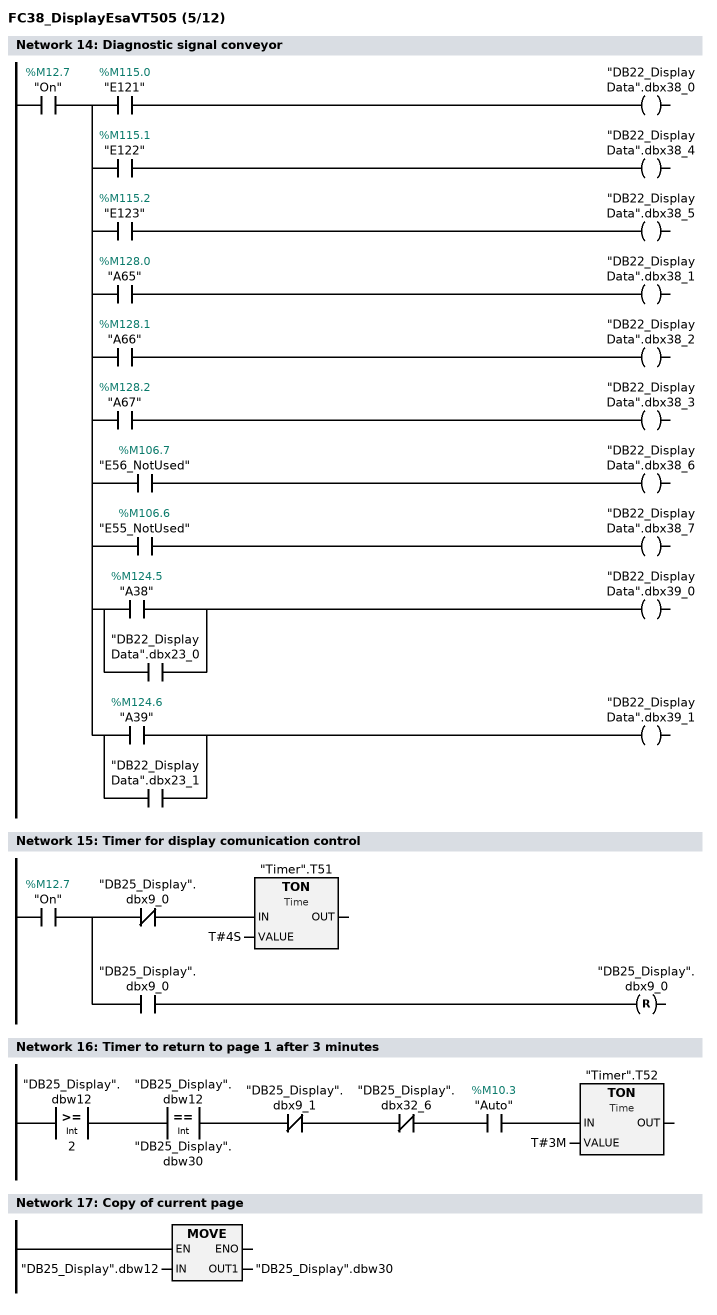
   RUNG wire#powerrail
      Contact( "On" )
      wire#w1
      Contact( "E121" )
      Coil( "DB22_DisplayData".dbx38_0 )
   END_RUNG
   RUNG wire#w1
      Contact( "E122" )
      Coil( "DB22_DisplayData".dbx38_4 )
   END_RUNG
   RUNG wire#w1
      Contact( "E123" )
      Coil( "DB22_DisplayData".dbx38_5 )
   END_RUNG
   RUNG wire#w1
      Contact( "A65" )
      Coil( "DB22_DisplayData".dbx38_1 )
   END_RUNG
   RUNG wire#w1
      Contact( "A66" )
      Coil( "DB22_DisplayData".dbx38_2 )
   END_RUNG
   RUNG wire#w1
      Contact( "A67" )
      Coil( "DB22_DisplayData".dbx38_3 )
   END_RUNG
   RUNG wire#w1
      Contact( "E56_NotUsed" )
      Coil( "DB22_DisplayData".dbx38_6 )
   END_RUNG
   RUNG wire#w1
      Contact( "E55_NotUsed" )
      Coil( "DB22_DisplayData".dbx38_7 )
   END_RUNG
   RUNG wire#w1
      Contact( "A38" )
      wire#w2
      Coil( "DB22_DisplayData".dbx39_0 )
   END_RUNG
   RUNG wire#w1
      Contact( "DB22_DisplayData".dbx23_0 )
   END_RUNG wire#w2
   RUNG wire#w1
      Contact( "A39" )
      wire#w3
      Coil( "DB22_DisplayData".dbx39_1 )
   END_RUNG
   RUNG wire#w1
      Contact( "DB22_DisplayData".dbx23_1 )
   END_RUNG wire#w3
   // the same network as SCL:
   "DB22_DisplayData".dbx38_0 := "On" AND "E121";
   "DB22_DisplayData".dbx38_4 := "On" AND "E122";
   "DB22_DisplayData".dbx38_5 := "On" AND "E123";
   "DB22_DisplayData".dbx38_1 := "On" AND "A65";
   "DB22_DisplayData".dbx38_2 := "On" AND "A66";
   "DB22_DisplayData".dbx38_3 := "On" AND "A67";
   "DB22_DisplayData".dbx38_6 := "On" AND "E56_NotUsed";
   "DB22_DisplayData".dbx38_7 := "On" AND "E55_NotUsed";
   "DB22_DisplayData".dbx39_0 := "On" AND ("A38" OR "DB22_DisplayData".dbx23_0);
   "DB22_DisplayData".dbx39_1 := "On" AND ("A39" OR "DB22_DisplayData".dbx23_1);
END_REGION

REGION Network 15: Timer for display comunication control
   "Timer".T51.TON(IN := "On" AND NOT "DB25_Display".dbx9_0, PT := T#4S);   // TON coil
   IF "On" AND "DB25_Display".dbx9_0 THEN "DB25_Display".dbx9_0 := FALSE; END_IF;
END_REGION

REGION Network 16: Timer to return to page 1 after 3 minutes
   "Timer".T52.TON(IN := ("DB25_Display".dbw12 >= 2) AND ("DB25_Display".dbw12 = "DB25_Display".dbw30) AND NOT "DB25_Display".dbx9_1 AND NOT "DB25_Display".dbx32_6 AND "Auto", PT := T#3M);   // TON coil
END_REGION

REGION Network 17: Copy of current page
   RUNG wire#powerrail
      { S7_GenerateENO := "TRUE" } Move(in := "DB25_Display".dbw12, out1 => "DB25_Display".dbw30)
   END_RUNG
   // the same network as SCL:
   "DB25_Display".dbw30 := "DB25_Display".dbw12;
END_REGION

REGION Network 18: Return to page 1 after 3 minutes
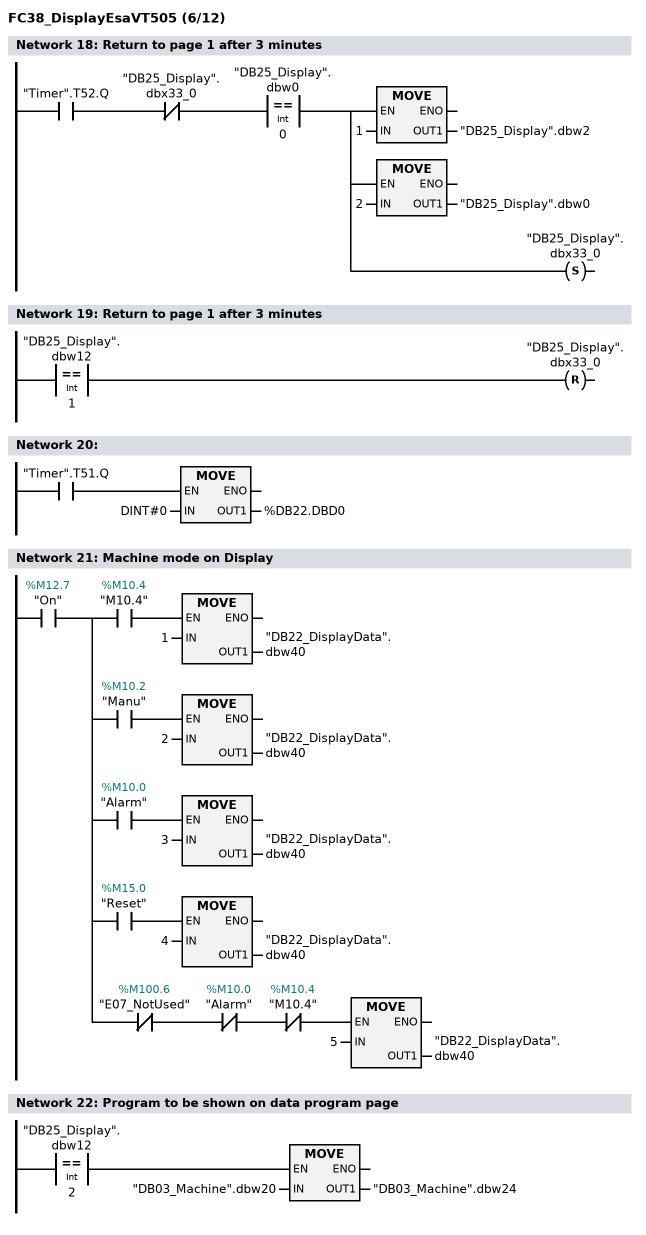
   RUNG wire#powerrail
      Contact( "Timer".T52.Q )
      I_Contact( "DB25_Display".dbx33_0 )
      { S7_Templates := "SrcType := Int" } EQ_Contact(in1 := "DB25_Display".dbw0, in2 := 0)
      wire#w1
      { S7_GenerateENO := "TRUE" } Move(in := 1, out1 => "DB25_Display".dbw2)
   END_RUNG
   RUNG wire#w1
      { S7_GenerateENO := "TRUE" } Move(in := 2, out1 => "DB25_Display".dbw0)
   END_RUNG
   RUNG wire#w1
      S_Coil( "DB25_Display".dbx33_0 )
   END_RUNG
   // the same network as SCL:
   IF "Timer".T52.Q AND NOT "DB25_Display".dbx33_0 AND ("DB25_Display".dbw0 = 0) THEN
       "DB25_Display".dbw2 := 1;
   END_IF;
   #_w1 := "Timer".T52.Q AND NOT "DB25_Display".dbx33_0 AND ("DB25_Display".dbw0 = 0);
   IF #_w1 THEN
       "DB25_Display".dbw0 := 2;
       "DB25_Display".dbx33_0 := TRUE;
   END_IF;
END_REGION

REGION Network 19: Return to page 1 after 3 minutes
   RUNG wire#powerrail
      { S7_Templates := "SrcType := Int" } EQ_Contact(in1 := "DB25_Display".dbw12, in2 := 1)
      R_Coil( "DB25_Display".dbx33_0 )
   END_RUNG
   // the same network as SCL:
   IF "DB25_Display".dbw12 = 1 THEN "DB25_Display".dbx33_0 := FALSE; END_IF;
END_REGION

REGION Network 20
   RUNG wire#powerrail
      Contact( "Timer".T51.Q )
      { S7_GenerateENO := "TRUE" } Move(in := DINT#0, out1 => %DB22.DBD0)
   END_RUNG
   // the same network as SCL:
   IF "Timer".T51.Q THEN %DB22.DBD0 := DINT#0; END_IF;
END_REGION

REGION Network 21: Machine mode on Display
   RUNG wire#powerrail
      Contact( "On" )
      wire#w1
      Contact( "M10.4" )
      { S7_GenerateENO := "TRUE" } Move(in := 1, out1 => "DB22_DisplayData".dbw40)
   END_RUNG
   RUNG wire#w1
      Contact( "Manu" )
      { S7_GenerateENO := "TRUE" } Move(in := 2, out1 => "DB22_DisplayData".dbw40)
   END_RUNG
   RUNG wire#w1
      Contact( "Alarm" )
      { S7_GenerateENO := "TRUE" } Move(in := 3, out1 => "DB22_DisplayData".dbw40)
   END_RUNG
   RUNG wire#w1
      Contact( "Reset" )
      { S7_GenerateENO := "TRUE" } Move(in := 4, out1 => "DB22_DisplayData".dbw40)
   END_RUNG
   RUNG wire#w1
      I_Contact( "E07_NotUsed" )
      I_Contact( "Alarm" )
      I_Contact( "M10.4" )
      { S7_GenerateENO := "TRUE" } Move(in := 5, out1 => "DB22_DisplayData".dbw40)
   END_RUNG
   // the same network as SCL:
   IF "On" AND "M10.4" THEN "DB22_DisplayData".dbw40 := 1; END_IF;
   IF "On" AND "Manu" THEN "DB22_DisplayData".dbw40 := 2; END_IF;
   IF "On" AND "Alarm" THEN "DB22_DisplayData".dbw40 := 3; END_IF;
   IF "On" AND "Reset" THEN "DB22_DisplayData".dbw40 := 4; END_IF;
   IF "On" AND NOT "E07_NotUsed" AND NOT "Alarm" AND NOT "M10.4" THEN "DB22_DisplayData".dbw40 := 5; END_IF;
END_REGION

REGION Network 22: Program to be shown on data program page
   RUNG wire#powerrail
      { S7_Templates := "SrcType := Int" } EQ_Contact(in1 := "DB25_Display".dbw12, in2 := 2)
      { S7_GenerateENO := "TRUE" } Move(in := "DB03_Machine".dbw20, out1 => "DB03_Machine".dbw24)
   END_RUNG
   // the same network as SCL:
   IF "DB25_Display".dbw12 = 2 THEN "DB03_Machine".dbw24 := "DB03_Machine".dbw20; END_IF;
END_REGION

REGION Network 23: Load data from data table to display area
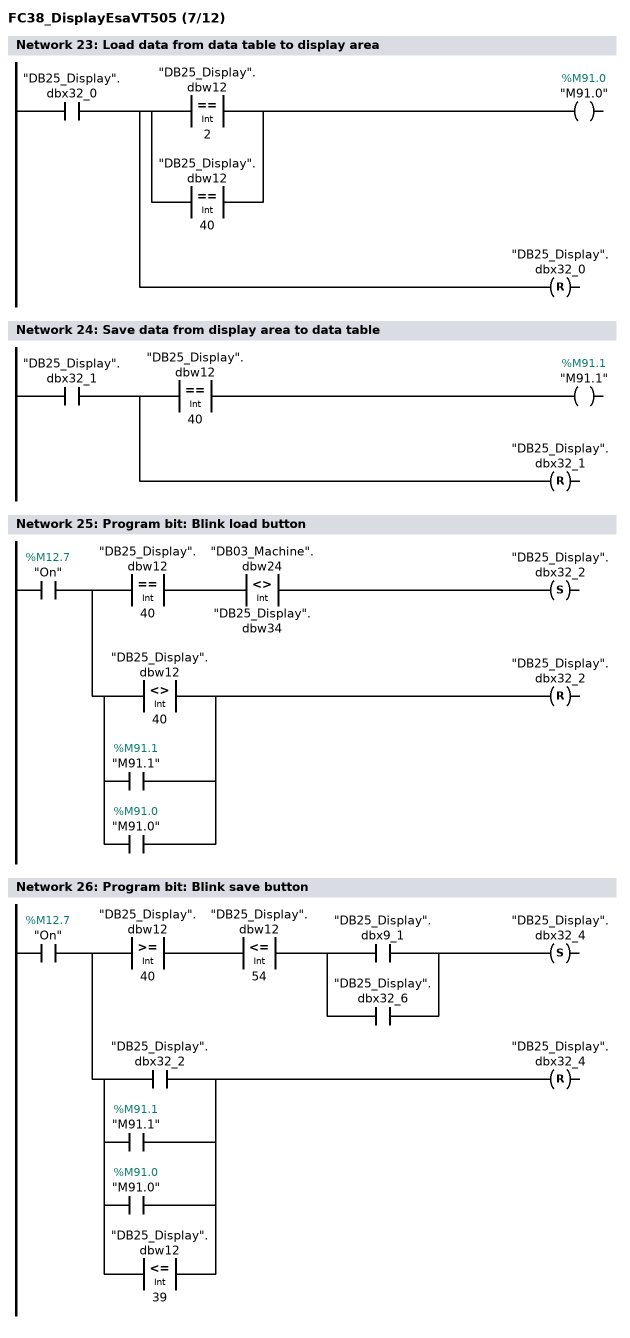
   RUNG wire#powerrail
      Contact( "DB25_Display".dbx32_0 )
      wire#w1
      { S7_Templates := "SrcType := Int" } EQ_Contact(in1 := "DB25_Display".dbw12, in2 := 2)
      wire#w2
      Coil( "M91.0" )
   END_RUNG
   RUNG wire#w1
      { S7_Templates := "SrcType := Int" } EQ_Contact(in1 := "DB25_Display".dbw12, in2 := 40)
   END_RUNG wire#w2
   RUNG wire#w1
      R_Coil( "DB25_Display".dbx32_0 )
   END_RUNG
   // the same network as SCL:
   "M91.0" := "DB25_Display".dbx32_0 AND (("DB25_Display".dbw12 = 2) OR ("DB25_Display".dbw12 = 40));
   IF "DB25_Display".dbx32_0 THEN "DB25_Display".dbx32_0 := FALSE; END_IF;
END_REGION

REGION Network 24: Save data from display area to data table
   RUNG wire#powerrail
      Contact( "DB25_Display".dbx32_1 )
      wire#w1
      { S7_Templates := "SrcType := Int" } EQ_Contact(in1 := "DB25_Display".dbw12, in2 := 40)
      Coil( "M91.1" )
   END_RUNG
   RUNG wire#w1
      R_Coil( "DB25_Display".dbx32_1 )
   END_RUNG
   // the same network as SCL:
   "M91.1" := "DB25_Display".dbx32_1 AND ("DB25_Display".dbw12 = 40);
   IF "DB25_Display".dbx32_1 THEN "DB25_Display".dbx32_1 := FALSE; END_IF;
END_REGION

REGION Network 25: Program bit: Blink load button
   RUNG wire#powerrail
      Contact( "On" )
      wire#w1
      { S7_Templates := "SrcType := Int" } EQ_Contact(in1 := "DB25_Display".dbw12, in2 := 40)
      { S7_Templates := "SrcType := Int" } NE_Contact(in1 := "DB03_Machine".dbw24, in2 := "DB25_Display".dbw34)
      S_Coil( "DB25_Display".dbx32_2 )
   END_RUNG
   RUNG wire#w1
      { S7_Templates := "SrcType := Int" } NE_Contact(in1 := "DB25_Display".dbw12, in2 := 40)
      wire#w2
      R_Coil( "DB25_Display".dbx32_2 )
   END_RUNG
   RUNG wire#w1
      Contact( "M91.1" )
   END_RUNG wire#w2
   RUNG wire#w1
      Contact( "M91.0" )
   END_RUNG wire#w2
   // the same network as SCL:
   IF "On" AND ("DB25_Display".dbw12 = 40) AND ("DB03_Machine".dbw24 <> "DB25_Display".dbw34) THEN
       "DB25_Display".dbx32_2 := TRUE;
   END_IF;
   IF "On" AND (("DB25_Display".dbw12 <> 40) OR "M91.1" OR "M91.0") THEN
       "DB25_Display".dbx32_2 := FALSE;
   END_IF;
END_REGION

REGION Network 26: Program bit: Blink save button
   RUNG wire#powerrail
      Contact( "On" )
      wire#w1
      { S7_Templates := "SrcType := Int" } GE_Contact(in1 := "DB25_Display".dbw12, in2 := 40)
      { S7_Templates := "SrcType := Int" } LE_Contact(in1 := "DB25_Display".dbw12, in2 := 54)
      wire#w2
      Contact( "DB25_Display".dbx9_1 )
      wire#w3
      S_Coil( "DB25_Display".dbx32_4 )
   END_RUNG
   RUNG wire#w2
      Contact( "DB25_Display".dbx32_6 )
   END_RUNG wire#w3
   RUNG wire#w1
      Contact( "DB25_Display".dbx32_2 )
      wire#w4
      R_Coil( "DB25_Display".dbx32_4 )
   END_RUNG
   RUNG wire#w1
      Contact( "M91.1" )
   END_RUNG wire#w4
   RUNG wire#w1
      Contact( "M91.0" )
   END_RUNG wire#w4
   RUNG wire#w1
      { S7_Templates := "SrcType := Int" } LE_Contact(in1 := "DB25_Display".dbw12, in2 := 39)
   END_RUNG wire#w4
   // the same network as SCL:
   IF "On" AND ("DB25_Display".dbw12 >= 40) AND ("DB25_Display".dbw12 <= 54) AND ("DB25_Display".dbx9_1 OR "DB25_Display".dbx32_6) THEN
       "DB25_Display".dbx32_4 := TRUE;
   END_IF;
   IF "On" AND ("DB25_Display".dbx32_2 OR "M91.1" OR "M91.0" OR ("DB25_Display".dbw12 <= 39)) THEN
       "DB25_Display".dbx32_4 := FALSE;
   END_IF;
END_REGION

REGION Network 27: Program bit:Blink load and save button
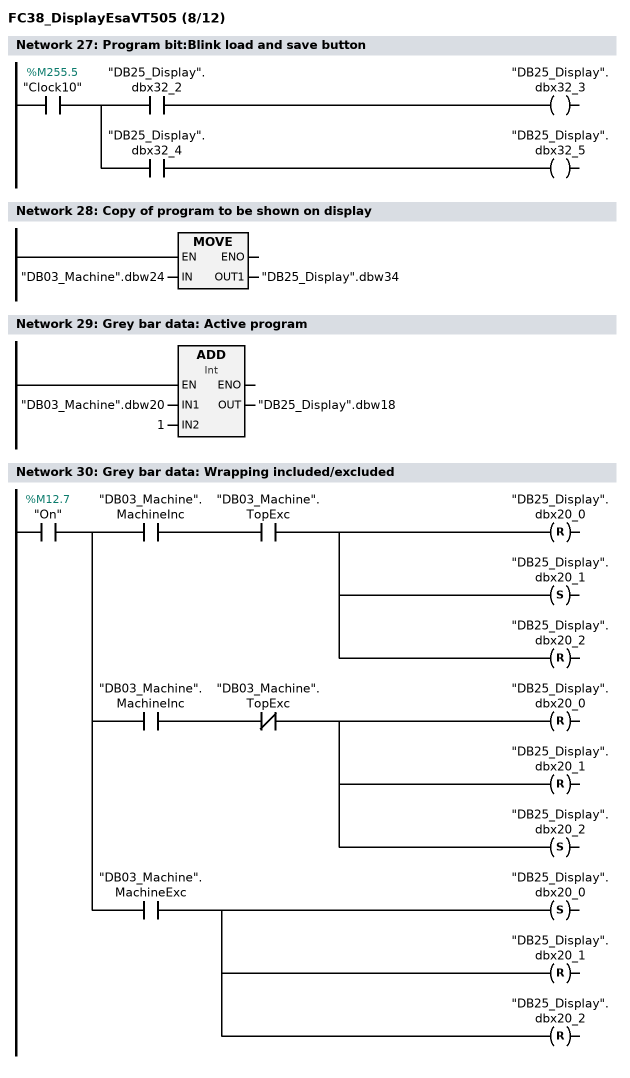
   RUNG wire#powerrail
      Contact( "Clock10" )
      wire#w1
      Contact( "DB25_Display".dbx32_2 )
      Coil( "DB25_Display".dbx32_3 )
   END_RUNG
   RUNG wire#w1
      Contact( "DB25_Display".dbx32_4 )
      Coil( "DB25_Display".dbx32_5 )
   END_RUNG
   // the same network as SCL:
   "DB25_Display".dbx32_3 := "Clock10" AND "DB25_Display".dbx32_2;
   "DB25_Display".dbx32_5 := "Clock10" AND "DB25_Display".dbx32_4;
END_REGION

REGION Network 28: Copy of program to be shown on display
   RUNG wire#powerrail
      { S7_GenerateENO := "TRUE" } Move(in := "DB03_Machine".dbw24, out1 => "DB25_Display".dbw34)
   END_RUNG
   // the same network as SCL:
   "DB25_Display".dbw34 := "DB03_Machine".dbw24;
END_REGION

REGION Network 29: Grey bar data: Active program
   RUNG wire#powerrail
      { S7_Templates := "SrcType := Int"; S7_GenerateENO := "TRUE" } Add(in1 := "DB03_Machine".dbw20, in2 := 1, out => "DB25_Display".dbw18)
   END_RUNG
   // the same network as SCL:
   "DB25_Display".dbw18 := "DB03_Machine".dbw20 + 1;
END_REGION

REGION Network 30: Grey bar data: Wrapping included/excluded
   RUNG wire#powerrail
      Contact( "On" )
      wire#w1
      Contact( "DB03_Machine".MachineInc )
      Contact( "DB03_Machine".TopExc )
      wire#w2
      R_Coil( "DB25_Display".dbx20_0 )
   END_RUNG
   RUNG wire#w2
      S_Coil( "DB25_Display".dbx20_1 )
   END_RUNG
   RUNG wire#w2
      R_Coil( "DB25_Display".dbx20_2 )
   END_RUNG
   RUNG wire#w1
      Contact( "DB03_Machine".MachineInc )
      I_Contact( "DB03_Machine".TopExc )
      wire#w3
      R_Coil( "DB25_Display".dbx20_0 )
   END_RUNG
   RUNG wire#w3
      R_Coil( "DB25_Display".dbx20_1 )
   END_RUNG
   RUNG wire#w3
      S_Coil( "DB25_Display".dbx20_2 )
   END_RUNG
   RUNG wire#w1
      Contact( "DB03_Machine".MachineExc )
      wire#w4
      S_Coil( "DB25_Display".dbx20_0 )
   END_RUNG
   RUNG wire#w4
      R_Coil( "DB25_Display".dbx20_1 )
   END_RUNG
   RUNG wire#w4
      R_Coil( "DB25_Display".dbx20_2 )
   END_RUNG
   // the same network as SCL:
   IF "On" AND "DB03_Machine".MachineInc AND "DB03_Machine".TopExc THEN
       "DB25_Display".dbx20_0 := FALSE;
       "DB25_Display".dbx20_1 := TRUE;
       "DB25_Display".dbx20_2 := FALSE;
   END_IF;
   IF "On" AND "DB03_Machine".MachineInc AND NOT "DB03_Machine".TopExc THEN
       "DB25_Display".dbx20_0 := FALSE;
       "DB25_Display".dbx20_1 := FALSE;
       "DB25_Display".dbx20_2 := TRUE;
   END_IF;
   IF "On" AND "DB03_Machine".MachineExc THEN
       "DB25_Display".dbx20_0 := TRUE;
       "DB25_Display".dbx20_1 := FALSE;
       "DB25_Display".dbx20_2 := FALSE;
   END_IF;
END_REGION

REGION Network 31: Grey bar data: Pressure plate included/excluded
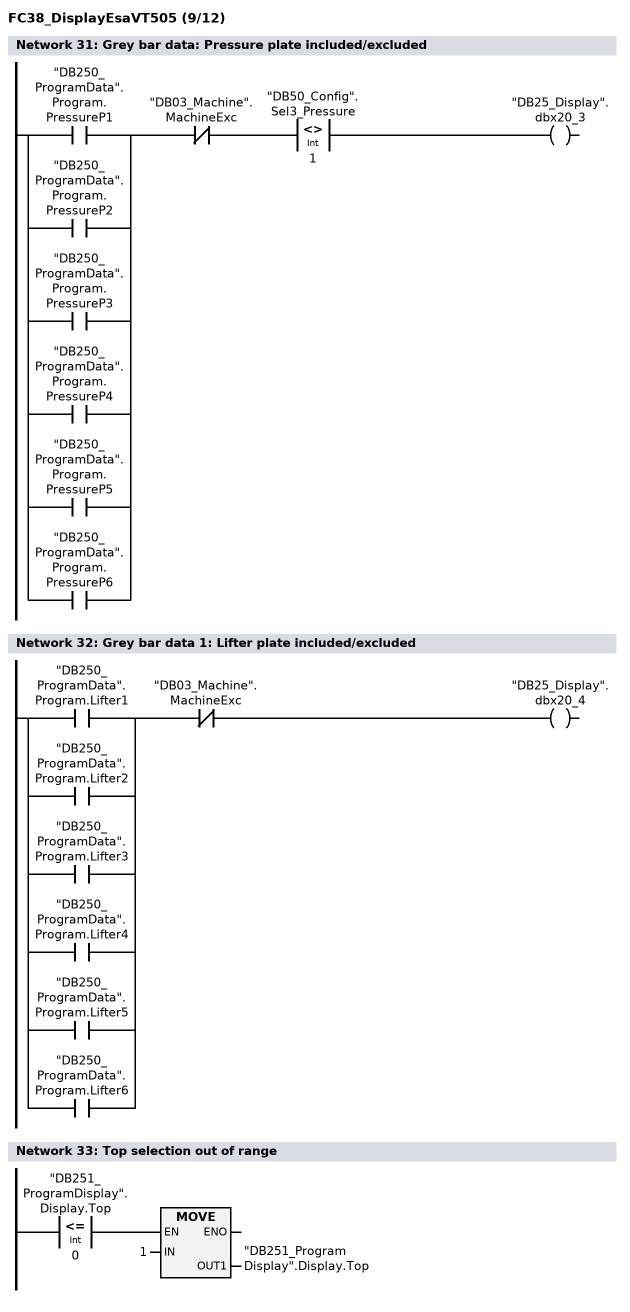
   RUNG wire#powerrail
      Contact( "DB250_ProgramData".Program.PressureP1 )
      wire#w1
      I_Contact( "DB03_Machine".MachineExc )
      { S7_Templates := "SrcType := Int" } NE_Contact(in1 := "DB50_Config".Sel3_Pressure, in2 := 1)
      Coil( "DB25_Display".dbx20_3 )
   END_RUNG
   RUNG wire#powerrail
      Contact( "DB250_ProgramData".Program.PressureP2 )
   END_RUNG wire#w1
   RUNG wire#powerrail
      Contact( "DB250_ProgramData".Program.PressureP3 )
   END_RUNG wire#w1
   RUNG wire#powerrail
      Contact( "DB250_ProgramData".Program.PressureP4 )
   END_RUNG wire#w1
   RUNG wire#powerrail
      Contact( "DB250_ProgramData".Program.PressureP5 )
   END_RUNG wire#w1
   RUNG wire#powerrail
      Contact( "DB250_ProgramData".Program.PressureP6 )
   END_RUNG wire#w1
   // the same network as SCL:
   "DB25_Display".dbx20_3 := ("DB250_ProgramData".Program.PressureP1 OR "DB250_ProgramData".Program.PressureP2 OR "DB250_ProgramData".Program.PressureP3 OR "DB250_ProgramData".Program.PressureP4 OR "DB250_ProgramData".Program.PressureP5 OR "DB250_ProgramData".Program.PressureP6) AND NOT "DB03_Machine".MachineExc AND ("DB50_Config".Sel3_Pressure <> 1);
END_REGION

REGION Network 32: Grey bar data 1: Lifter plate included/excluded
   RUNG wire#powerrail
      Contact( "DB250_ProgramData".Program.Lifter1 )
      wire#w1
      I_Contact( "DB03_Machine".MachineExc )
      Coil( "DB25_Display".dbx20_4 )
   END_RUNG
   RUNG wire#powerrail
      Contact( "DB250_ProgramData".Program.Lifter2 )
   END_RUNG wire#w1
   RUNG wire#powerrail
      Contact( "DB250_ProgramData".Program.Lifter3 )
   END_RUNG wire#w1
   RUNG wire#powerrail
      Contact( "DB250_ProgramData".Program.Lifter4 )
   END_RUNG wire#w1
   RUNG wire#powerrail
      Contact( "DB250_ProgramData".Program.Lifter5 )
   END_RUNG wire#w1
   RUNG wire#powerrail
      Contact( "DB250_ProgramData".Program.Lifter6 )
   END_RUNG wire#w1
   // the same network as SCL:
   "DB25_Display".dbx20_4 := ("DB250_ProgramData".Program.Lifter1 OR "DB250_ProgramData".Program.Lifter2 OR "DB250_ProgramData".Program.Lifter3 OR "DB250_ProgramData".Program.Lifter4 OR "DB250_ProgramData".Program.Lifter5 OR "DB250_ProgramData".Program.Lifter6) AND NOT "DB03_Machine".MachineExc;
END_REGION

REGION Network 33: Top selection out of range
   RUNG wire#powerrail
      { S7_Templates := "SrcType := Int" } LE_Contact(in1 := "DB251_ProgramDisplay".Display.Top, in2 := 0)
      { S7_GenerateENO := "TRUE" } Move(in := 1, out1 => "DB251_ProgramDisplay".Display.Top)
   END_RUNG
   // the same network as SCL:
   IF "DB251_ProgramDisplay".Display.Top <= 0 THEN "DB251_ProgramDisplay".Display.Top := 1; END_IF;
END_REGION

REGION Network 34: Top film lenght out of range
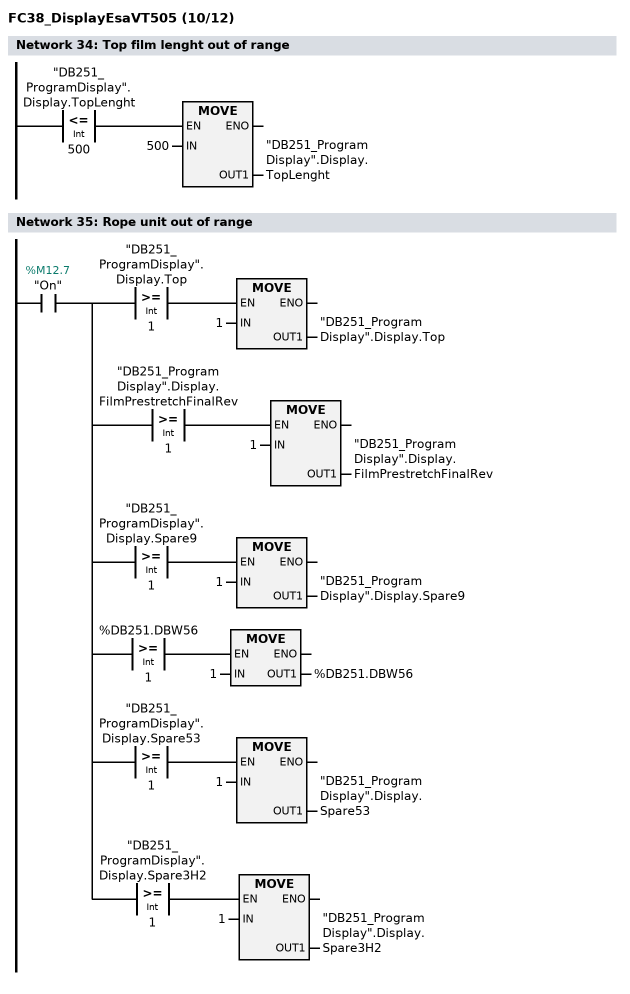
   RUNG wire#powerrail
      { S7_Templates := "SrcType := Int" } LE_Contact(in1 := "DB251_ProgramDisplay".Display.TopLenght, in2 := 500)
      { S7_GenerateENO := "TRUE" } Move(in := 500, out1 => "DB251_ProgramDisplay".Display.TopLenght)
   END_RUNG
   // the same network as SCL:
   IF "DB251_ProgramDisplay".Display.TopLenght <= 500 THEN
       "DB251_ProgramDisplay".Display.TopLenght := 500;
   END_IF;
END_REGION

REGION Network 35: Rope unit out of range
   RUNG wire#powerrail
      Contact( "On" )
      wire#w1
      { S7_Templates := "SrcType := Int" } GE_Contact(in1 := "DB251_ProgramDisplay".Display.Top, in2 := 1)
      { S7_GenerateENO := "TRUE" } Move(in := 1, out1 => "DB251_ProgramDisplay".Display.Top)
   END_RUNG
   RUNG wire#w1
      { S7_Templates := "SrcType := Int" } GE_Contact(in1 := "DB251_ProgramDisplay".Display.FilmPrestretchFinalRev, in2 := 1)
      { S7_GenerateENO := "TRUE" } Move(in := 1, out1 => "DB251_ProgramDisplay".Display.FilmPrestretchFinalRev)
   END_RUNG
   RUNG wire#w1
      { S7_Templates := "SrcType := Int" } GE_Contact(in1 := "DB251_ProgramDisplay".Display.Spare9, in2 := 1)
      { S7_GenerateENO := "TRUE" } Move(in := 1, out1 => "DB251_ProgramDisplay".Display.Spare9)
   END_RUNG
   RUNG wire#w1
      { S7_Templates := "SrcType := Int" } GE_Contact(in1 := %DB251.DBW56, in2 := 1)
      { S7_GenerateENO := "TRUE" } Move(in := 1, out1 => %DB251.DBW56)
   END_RUNG
   RUNG wire#w1
      { S7_Templates := "SrcType := Int" } GE_Contact(in1 := "DB251_ProgramDisplay".Display.Spare53, in2 := 1)
      { S7_GenerateENO := "TRUE" } Move(in := 1, out1 => "DB251_ProgramDisplay".Display.Spare53)
   END_RUNG
   RUNG wire#w1
      { S7_Templates := "SrcType := Int" } GE_Contact(in1 := "DB251_ProgramDisplay".Display.Spare3H2, in2 := 1)
      { S7_GenerateENO := "TRUE" } Move(in := 1, out1 => "DB251_ProgramDisplay".Display.Spare3H2)
   END_RUNG
   // the same network as SCL:
   IF "On" AND ("DB251_ProgramDisplay".Display.Top >= 1) THEN
       "DB251_ProgramDisplay".Display.Top := 1;
   END_IF;
   IF "On" AND ("DB251_ProgramDisplay".Display.FilmPrestretchFinalRev >= 1) THEN
       "DB251_ProgramDisplay".Display.FilmPrestretchFinalRev := 1;
   END_IF;
   IF "On" AND ("DB251_ProgramDisplay".Display.Spare9 >= 1) THEN
       "DB251_ProgramDisplay".Display.Spare9 := 1;
   END_IF;
   IF "On" AND (%DB251.DBW56 >= 1) THEN %DB251.DBW56 := 1; END_IF;
   IF "On" AND ("DB251_ProgramDisplay".Display.Spare53 >= 1) THEN
       "DB251_ProgramDisplay".Display.Spare53 := 1;
   END_IF;
   IF "On" AND ("DB251_ProgramDisplay".Display.Spare3H2 >= 1) THEN
       "DB251_ProgramDisplay".Display.Spare3H2 := 1;
   END_IF;
END_REGION

REGION Network 36: Rope unit out of range
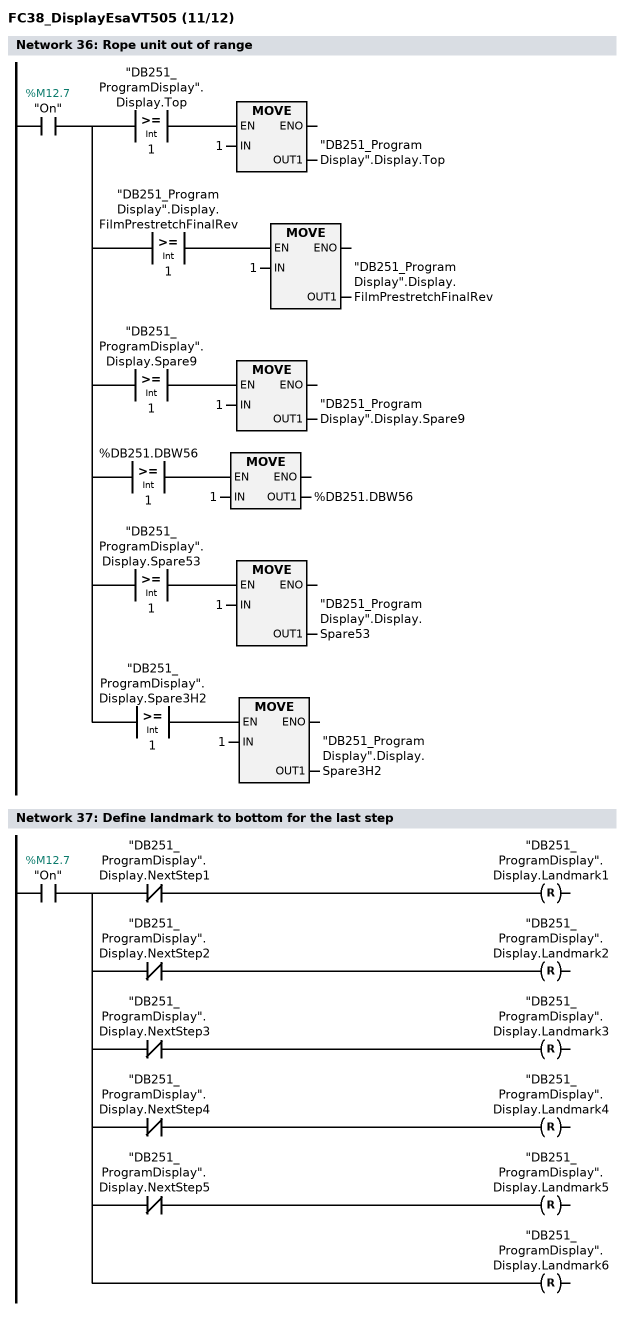
   RUNG wire#powerrail
      Contact( "On" )
      wire#w1
      { S7_Templates := "SrcType := Int" } GE_Contact(in1 := "DB251_ProgramDisplay".Display.Top, in2 := 1)
      { S7_GenerateENO := "TRUE" } Move(in := 1, out1 => "DB251_ProgramDisplay".Display.Top)
   END_RUNG
   RUNG wire#w1
      { S7_Templates := "SrcType := Int" } GE_Contact(in1 := "DB251_ProgramDisplay".Display.FilmPrestretchFinalRev, in2 := 1)
      { S7_GenerateENO := "TRUE" } Move(in := 1, out1 => "DB251_ProgramDisplay".Display.FilmPrestretchFinalRev)
   END_RUNG
   RUNG wire#w1
      { S7_Templates := "SrcType := Int" } GE_Contact(in1 := "DB251_ProgramDisplay".Display.Spare9, in2 := 1)
      { S7_GenerateENO := "TRUE" } Move(in := 1, out1 => "DB251_ProgramDisplay".Display.Spare9)
   END_RUNG
   RUNG wire#w1
      { S7_Templates := "SrcType := Int" } GE_Contact(in1 := %DB251.DBW56, in2 := 1)
      { S7_GenerateENO := "TRUE" } Move(in := 1, out1 => %DB251.DBW56)
   END_RUNG
   RUNG wire#w1
      { S7_Templates := "SrcType := Int" } GE_Contact(in1 := "DB251_ProgramDisplay".Display.Spare53, in2 := 1)
      { S7_GenerateENO := "TRUE" } Move(in := 1, out1 => "DB251_ProgramDisplay".Display.Spare53)
   END_RUNG
   RUNG wire#w1
      { S7_Templates := "SrcType := Int" } GE_Contact(in1 := "DB251_ProgramDisplay".Display.Spare3H2, in2 := 1)
      { S7_GenerateENO := "TRUE" } Move(in := 1, out1 => "DB251_ProgramDisplay".Display.Spare3H2)
   END_RUNG
   // the same network as SCL:
   IF "On" AND ("DB251_ProgramDisplay".Display.Top >= 1) THEN
       "DB251_ProgramDisplay".Display.Top := 1;
   END_IF;
   IF "On" AND ("DB251_ProgramDisplay".Display.FilmPrestretchFinalRev >= 1) THEN
       "DB251_ProgramDisplay".Display.FilmPrestretchFinalRev := 1;
   END_IF;
   IF "On" AND ("DB251_ProgramDisplay".Display.Spare9 >= 1) THEN
       "DB251_ProgramDisplay".Display.Spare9 := 1;
   END_IF;
   IF "On" AND (%DB251.DBW56 >= 1) THEN %DB251.DBW56 := 1; END_IF;
   IF "On" AND ("DB251_ProgramDisplay".Display.Spare53 >= 1) THEN
       "DB251_ProgramDisplay".Display.Spare53 := 1;
   END_IF;
   IF "On" AND ("DB251_ProgramDisplay".Display.Spare3H2 >= 1) THEN
       "DB251_ProgramDisplay".Display.Spare3H2 := 1;
   END_IF;
END_REGION

REGION Network 37: Define landmark to bottom for the last step
   RUNG wire#powerrail
      Contact( "On" )
      wire#w1
      I_Contact( "DB251_ProgramDisplay".Display.NextStep1 )
      R_Coil( "DB251_ProgramDisplay".Display.Landmark1 )
   END_RUNG
   RUNG wire#w1
      I_Contact( "DB251_ProgramDisplay".Display.NextStep2 )
      R_Coil( "DB251_ProgramDisplay".Display.Landmark2 )
   END_RUNG
   RUNG wire#w1
      I_Contact( "DB251_ProgramDisplay".Display.NextStep3 )
      R_Coil( "DB251_ProgramDisplay".Display.Landmark3 )
   END_RUNG
   RUNG wire#w1
      I_Contact( "DB251_ProgramDisplay".Display.NextStep4 )
      R_Coil( "DB251_ProgramDisplay".Display.Landmark4 )
   END_RUNG
   RUNG wire#w1
      I_Contact( "DB251_ProgramDisplay".Display.NextStep5 )
      R_Coil( "DB251_ProgramDisplay".Display.Landmark5 )
   END_RUNG
   RUNG wire#w1
      R_Coil( "DB251_ProgramDisplay".Display.Landmark6 )
   END_RUNG
   // the same network as SCL:
   IF "On" AND NOT "DB251_ProgramDisplay".Display.NextStep1 THEN
       "DB251_ProgramDisplay".Display.Landmark1 := FALSE;
   END_IF;
   IF "On" AND NOT "DB251_ProgramDisplay".Display.NextStep2 THEN
       "DB251_ProgramDisplay".Display.Landmark2 := FALSE;
   END_IF;
   IF "On" AND NOT "DB251_ProgramDisplay".Display.NextStep3 THEN
       "DB251_ProgramDisplay".Display.Landmark3 := FALSE;
   END_IF;
   IF "On" AND NOT "DB251_ProgramDisplay".Display.NextStep4 THEN
       "DB251_ProgramDisplay".Display.Landmark4 := FALSE;
   END_IF;
   IF "On" AND NOT "DB251_ProgramDisplay".Display.NextStep5 THEN
       "DB251_ProgramDisplay".Display.Landmark5 := FALSE;
   END_IF;
   IF "On" THEN "DB251_ProgramDisplay".Display.Landmark6 := FALSE; END_IF;
END_REGION

REGION Network 38
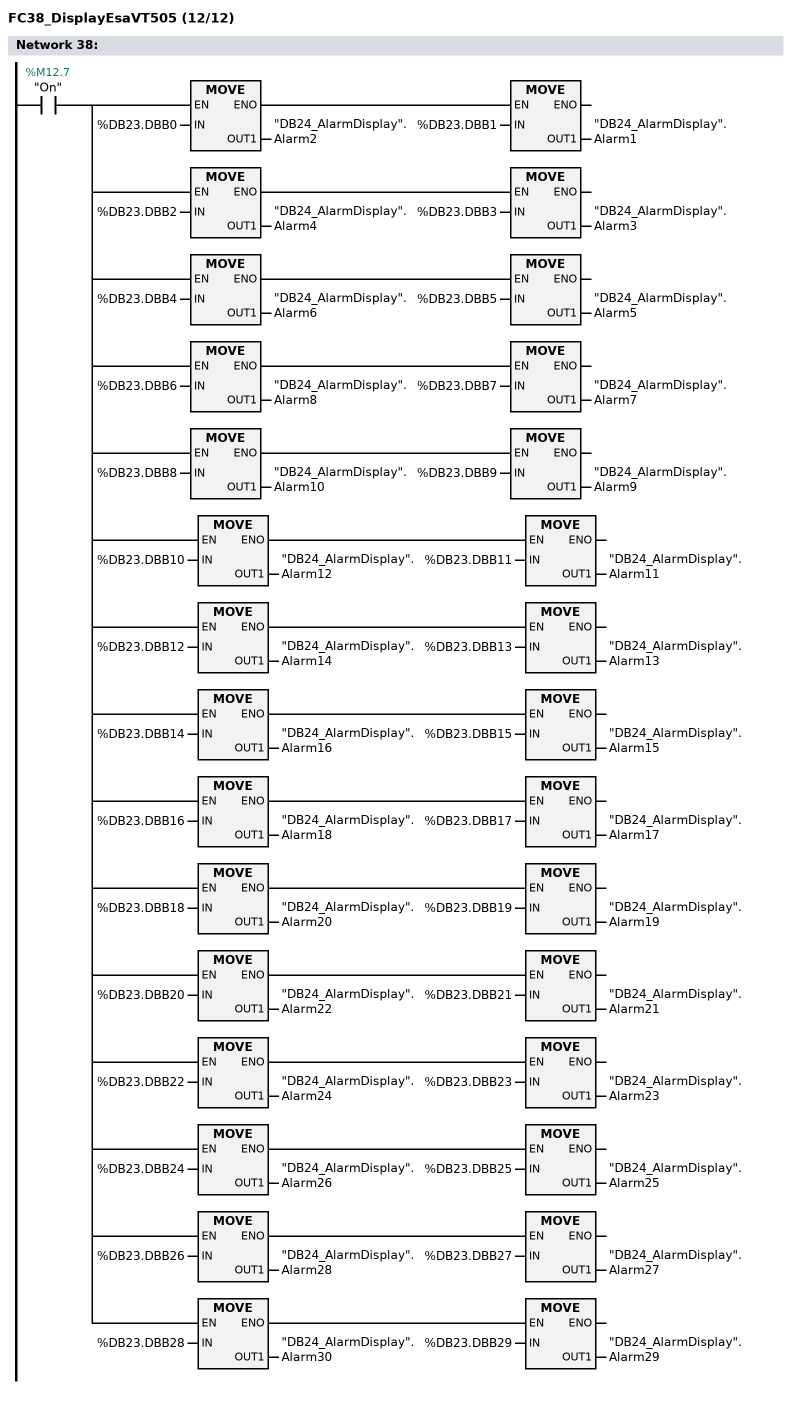
   RUNG wire#powerrail
      Contact( "On" )
      wire#w1
      { S7_GenerateENO := "TRUE" } Move(in := %DB23.DBB0, out1 => "DB24_AlarmDisplay".Alarm2)
      { S7_GenerateENO := "TRUE" } Move(in := %DB23.DBB1, out1 => "DB24_AlarmDisplay".Alarm1)
   END_RUNG
   RUNG wire#w1
      { S7_GenerateENO := "TRUE" } Move(in := %DB23.DBB2, out1 => "DB24_AlarmDisplay".Alarm4)
      { S7_GenerateENO := "TRUE" } Move(in := %DB23.DBB3, out1 => "DB24_AlarmDisplay".Alarm3)
   END_RUNG
   RUNG wire#w1
      { S7_GenerateENO := "TRUE" } Move(in := %DB23.DBB4, out1 => "DB24_AlarmDisplay".Alarm6)
      { S7_GenerateENO := "TRUE" } Move(in := %DB23.DBB5, out1 => "DB24_AlarmDisplay".Alarm5)
   END_RUNG
   RUNG wire#w1
      { S7_GenerateENO := "TRUE" } Move(in := %DB23.DBB6, out1 => "DB24_AlarmDisplay".Alarm8)
      { S7_GenerateENO := "TRUE" } Move(in := %DB23.DBB7, out1 => "DB24_AlarmDisplay".Alarm7)
   END_RUNG
   RUNG wire#w1
      { S7_GenerateENO := "TRUE" } Move(in := %DB23.DBB8, out1 => "DB24_AlarmDisplay".Alarm10)
      { S7_GenerateENO := "TRUE" } Move(in := %DB23.DBB9, out1 => "DB24_AlarmDisplay".Alarm9)
   END_RUNG
   RUNG wire#w1
      { S7_GenerateENO := "TRUE" } Move(in := %DB23.DBB10, out1 => "DB24_AlarmDisplay".Alarm12)
      { S7_GenerateENO := "TRUE" } Move(in := %DB23.DBB11, out1 => "DB24_AlarmDisplay".Alarm11)
   END_RUNG
   RUNG wire#w1
      { S7_GenerateENO := "TRUE" } Move(in := %DB23.DBB12, out1 => "DB24_AlarmDisplay".Alarm14)
      { S7_GenerateENO := "TRUE" } Move(in := %DB23.DBB13, out1 => "DB24_AlarmDisplay".Alarm13)
   END_RUNG
   RUNG wire#w1
      { S7_GenerateENO := "TRUE" } Move(in := %DB23.DBB14, out1 => "DB24_AlarmDisplay".Alarm16)
      { S7_GenerateENO := "TRUE" } Move(in := %DB23.DBB15, out1 => "DB24_AlarmDisplay".Alarm15)
   END_RUNG
   RUNG wire#w1
      { S7_GenerateENO := "TRUE" } Move(in := %DB23.DBB16, out1 => "DB24_AlarmDisplay".Alarm18)
      { S7_GenerateENO := "TRUE" } Move(in := %DB23.DBB17, out1 => "DB24_AlarmDisplay".Alarm17)
   END_RUNG
   RUNG wire#w1
      { S7_GenerateENO := "TRUE" } Move(in := %DB23.DBB18, out1 => "DB24_AlarmDisplay".Alarm20)
      { S7_GenerateENO := "TRUE" } Move(in := %DB23.DBB19, out1 => "DB24_AlarmDisplay".Alarm19)
   END_RUNG
   RUNG wire#w1
      { S7_GenerateENO := "TRUE" } Move(in := %DB23.DBB20, out1 => "DB24_AlarmDisplay".Alarm22)
      { S7_GenerateENO := "TRUE" } Move(in := %DB23.DBB21, out1 => "DB24_AlarmDisplay".Alarm21)
   END_RUNG
   RUNG wire#w1
      { S7_GenerateENO := "TRUE" } Move(in := %DB23.DBB22, out1 => "DB24_AlarmDisplay".Alarm24)
      { S7_GenerateENO := "TRUE" } Move(in := %DB23.DBB23, out1 => "DB24_AlarmDisplay".Alarm23)
   END_RUNG
   RUNG wire#w1
      { S7_GenerateENO := "TRUE" } Move(in := %DB23.DBB24, out1 => "DB24_AlarmDisplay".Alarm26)
      { S7_GenerateENO := "TRUE" } Move(in := %DB23.DBB25, out1 => "DB24_AlarmDisplay".Alarm25)
   END_RUNG
   RUNG wire#w1
      { S7_GenerateENO := "TRUE" } Move(in := %DB23.DBB26, out1 => "DB24_AlarmDisplay".Alarm28)
      { S7_GenerateENO := "TRUE" } Move(in := %DB23.DBB27, out1 => "DB24_AlarmDisplay".Alarm27)
   END_RUNG
   RUNG wire#w1
      { S7_GenerateENO := "TRUE" } Move(in := %DB23.DBB28, out1 => "DB24_AlarmDisplay".Alarm30)
      { S7_GenerateENO := "TRUE" } Move(in := %DB23.DBB29, out1 => "DB24_AlarmDisplay".Alarm29)
   END_RUNG
   // the same network as SCL:
   // ENO of a box is taken as its EN; it also drops when the box reports an error
   IF "On" THEN
       "DB24_AlarmDisplay".Alarm2 := %DB23.DBB0;
       "DB24_AlarmDisplay".Alarm1 := %DB23.DBB1;
       "DB24_AlarmDisplay".Alarm4 := %DB23.DBB2;
       "DB24_AlarmDisplay".Alarm3 := %DB23.DBB3;
       "DB24_AlarmDisplay".Alarm6 := %DB23.DBB4;
       "DB24_AlarmDisplay".Alarm5 := %DB23.DBB5;
       "DB24_AlarmDisplay".Alarm8 := %DB23.DBB6;
       "DB24_AlarmDisplay".Alarm7 := %DB23.DBB7;
       "DB24_AlarmDisplay".Alarm10 := %DB23.DBB8;
       "DB24_AlarmDisplay".Alarm9 := %DB23.DBB9;
       "DB24_AlarmDisplay".Alarm12 := %DB23.DBB10;
       "DB24_AlarmDisplay".Alarm11 := %DB23.DBB11;
       "DB24_AlarmDisplay".Alarm14 := %DB23.DBB12;
       "DB24_AlarmDisplay".Alarm13 := %DB23.DBB13;
       "DB24_AlarmDisplay".Alarm16 := %DB23.DBB14;
       "DB24_AlarmDisplay".Alarm15 := %DB23.DBB15;
       "DB24_AlarmDisplay".Alarm18 := %DB23.DBB16;
       "DB24_AlarmDisplay".Alarm17 := %DB23.DBB17;
       "DB24_AlarmDisplay".Alarm20 := %DB23.DBB18;
       "DB24_AlarmDisplay".Alarm19 := %DB23.DBB19;
       "DB24_AlarmDisplay".Alarm22 := %DB23.DBB20;
       "DB24_AlarmDisplay".Alarm21 := %DB23.DBB21;
       "DB24_AlarmDisplay".Alarm24 := %DB23.DBB22;
       "DB24_AlarmDisplay".Alarm23 := %DB23.DBB23;
       "DB24_AlarmDisplay".Alarm26 := %DB23.DBB24;
       "DB24_AlarmDisplay".Alarm25 := %DB23.DBB25;
       "DB24_AlarmDisplay".Alarm28 := %DB23.DBB26;
       "DB24_AlarmDisplay".Alarm27 := %DB23.DBB27;
       "DB24_AlarmDisplay".Alarm30 := %DB23.DBB28;
       "DB24_AlarmDisplay".Alarm29 := %DB23.DBB29;
   END_IF;
END_REGION
END_FUNCTION

FUNCTION "FC43_PreCarriageTechnoplat" : Void   // FC43, LAD
TITLE = HS40 standard prestretch management
{ S7_Optimized_Access := 'FALSE' }
AUTHOR : Robopac
VERSION : 0.0
// stored: AutoNumber false, IsIECCheckEnabled false, SetENOAutomatically false, UDAEnableTagReadback false
BEGIN

REGION Network 1: Timer for prestretch restart
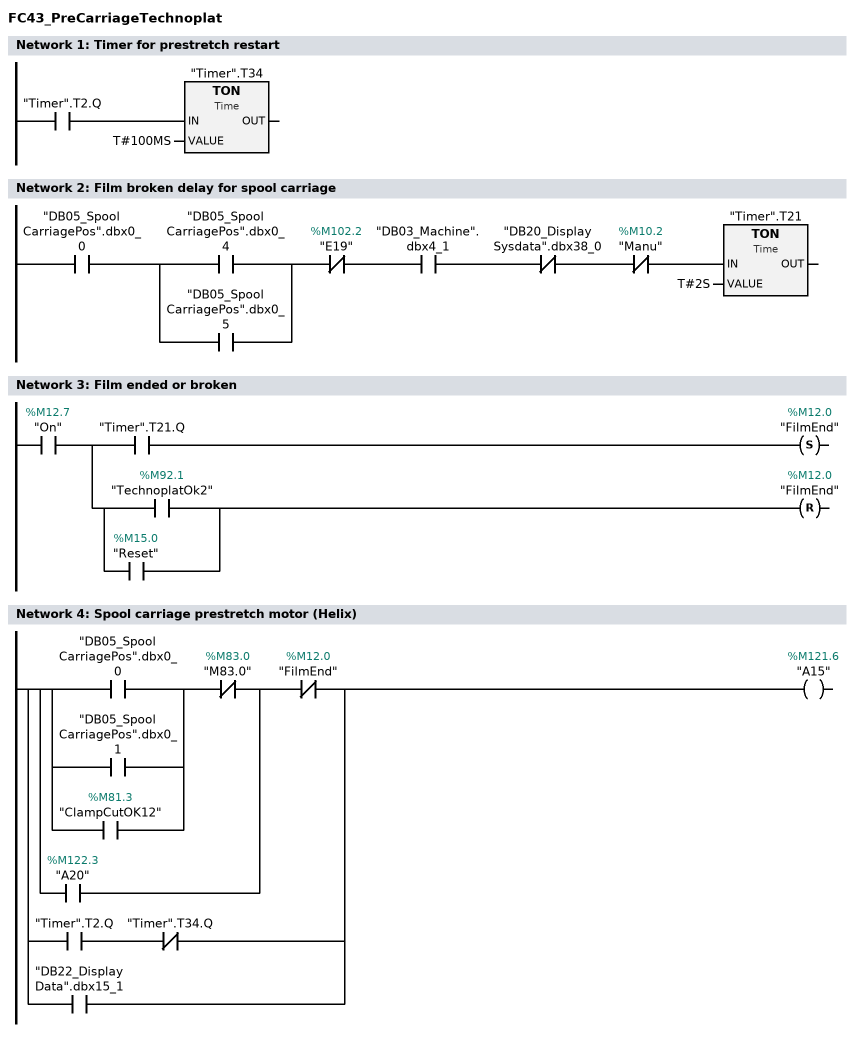
   "Timer".T34.TON(IN := "Timer".T2.Q, PT := T#100MS);   // TON coil
END_REGION

REGION Network 2: Film broken delay for spool carriage
   "Timer".T21.TON(IN := "DB05_SpoolCarriagePos".dbx0_0 AND ("DB05_SpoolCarriagePos".dbx0_4 OR "DB05_SpoolCarriagePos".dbx0_5) AND NOT "E19" AND "DB03_Machine".dbx4_1 AND NOT "DB20_DisplaySysdata".dbx38_0 AND NOT "Manu", PT := T#2S);   // TON coil
END_REGION

REGION Network 3: Film ended or broken
   RUNG wire#powerrail
      Contact( "On" )
      wire#w1
      Contact( "Timer".T21.Q )
      S_Coil( "FilmEnd" )
   END_RUNG
   RUNG wire#w1
      Contact( "TechnoplatOk2" )
      wire#w2
      R_Coil( "FilmEnd" )
   END_RUNG
   RUNG wire#w1
      Contact( "Reset" )
   END_RUNG wire#w2
   // the same network as SCL:
   IF "On" AND "Timer".T21.Q THEN "FilmEnd" := TRUE; END_IF;
   IF "On" AND ("TechnoplatOk2" OR "Reset") THEN "FilmEnd" := FALSE; END_IF;
END_REGION

REGION Network 4: Spool carriage prestretch motor (Helix)
   RUNG wire#powerrail
      Contact( "DB05_SpoolCarriagePos".dbx0_0 )
      wire#w1
      I_Contact( "M83.0" )
      wire#w2
      I_Contact( "FilmEnd" )
      wire#w3
      Coil( "A15" )
   END_RUNG
   RUNG wire#powerrail
      Contact( "DB05_SpoolCarriagePos".dbx0_1 )
   END_RUNG wire#w1
   RUNG wire#powerrail
      Contact( "ClampCutOK12" )
   END_RUNG wire#w1
   RUNG wire#powerrail
      Contact( "A20" )
   END_RUNG wire#w2
   RUNG wire#powerrail
      Contact( "Timer".T2.Q )
      I_Contact( "Timer".T34.Q )
   END_RUNG wire#w3
   RUNG wire#powerrail
      Contact( "DB22_DisplayData".dbx15_1 )
   END_RUNG wire#w3
   // the same network as SCL:
   "A15" := (((("DB05_SpoolCarriagePos".dbx0_0 OR "DB05_SpoolCarriagePos".dbx0_1 OR "ClampCutOK12") AND NOT "M83.0") OR "A20") AND NOT "FilmEnd") OR ("Timer".T2.Q AND NOT "Timer".T34.Q) OR "DB22_DisplayData".dbx15_1;
END_REGION
END_FUNCTION

FUNCTION "FC62_PreStretchPGSAoutPWM" : Void   // FC62, LAD
{ S7_Optimized_Access := 'FALSE' }
AUTHOR : PaZan
VERSION : 0.1
// stored: AutoNumber false, IsIECCheckEnabled false, SetENOAutomatically false, UDAEnableTagReadback false
BEGIN

REGION Network 1: copy parameter for scale value % prestretch
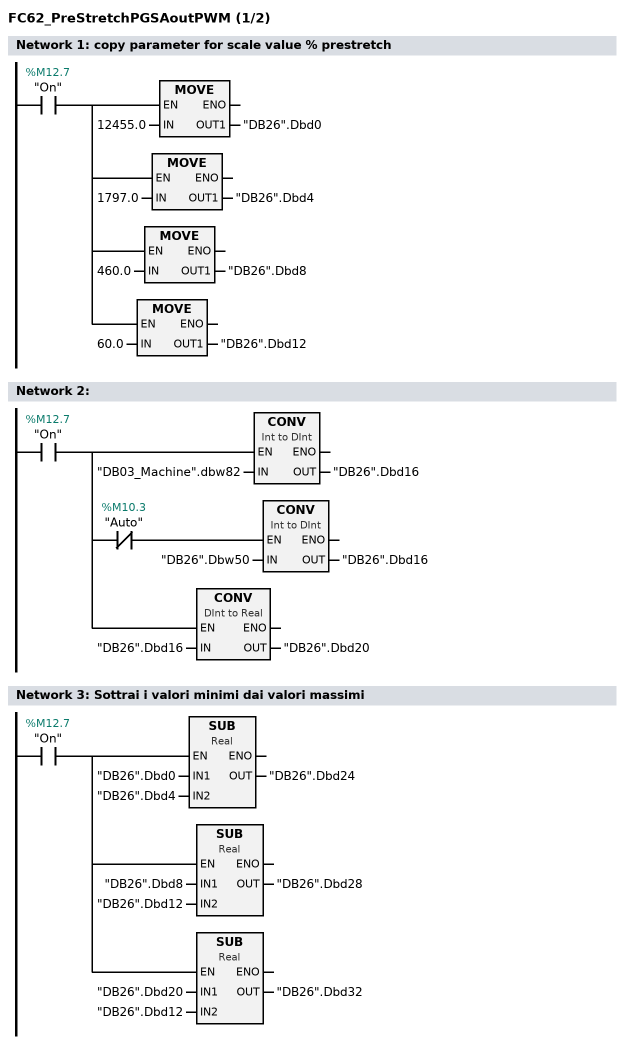
   RUNG wire#powerrail
      Contact( "On" )
      wire#w1
      { S7_GenerateENO := "TRUE" } Move(in := 12455.0, out1 => "DB26".Dbd0)
   END_RUNG
   RUNG wire#w1
      { S7_GenerateENO := "TRUE" } Move(in := 1797.0, out1 => "DB26".Dbd4)
   END_RUNG
   RUNG wire#w1
      { S7_GenerateENO := "TRUE" } Move(in := 460.0, out1 => "DB26".Dbd8)
   END_RUNG
   RUNG wire#w1
      { S7_GenerateENO := "TRUE" } Move(in := 60.0, out1 => "DB26".Dbd12)
   END_RUNG
   // the same network as SCL:
   IF "On" THEN
       "DB26".Dbd0 := 12455.0;
       "DB26".Dbd4 := 1797.0;
       "DB26".Dbd8 := 460.0;
       "DB26".Dbd12 := 60.0;
   END_IF;
END_REGION

REGION Network 2
   RUNG wire#powerrail
      Contact( "On" )
      wire#w1
      { S7_Templates := "[SrcType := Int, DestType := DInt]"; S7_GenerateENO := "TRUE" } Convert(in := "DB03_Machine".dbw82, out => "DB26".Dbd16)
   END_RUNG
   RUNG wire#w1
      I_Contact( "Auto" )
      { S7_Templates := "[SrcType := Int, DestType := DInt]"; S7_GenerateENO := "TRUE" } Convert(in := "DB26".Dbw50, out => "DB26".Dbd16)
   END_RUNG
   RUNG wire#w1
      { S7_Templates := "[SrcType := DInt, DestType := Real]"; S7_GenerateENO := "TRUE" } Convert(in := "DB26".Dbd16, out => "DB26".Dbd20)
   END_RUNG
   // the same network as SCL:
   IF "On" THEN "DB26".Dbd16 := INT_TO_DINT("DB03_Machine".dbw82); END_IF;
   IF "On" AND NOT "Auto" THEN "DB26".Dbd16 := INT_TO_DINT("DB26".Dbw50); END_IF;
   IF "On" THEN "DB26".Dbd20 := DINT_TO_REAL("DB26".Dbd16); END_IF;
END_REGION

REGION Network 3: Sottrai i valori minimi dai valori massimi
   RUNG wire#powerrail
      Contact( "On" )
      wire#w1
      { S7_Templates := "SrcType := Real"; S7_GenerateENO := "TRUE" } Sub(in1 := "DB26".Dbd0, in2 := "DB26".Dbd4, out => "DB26".Dbd24)
   END_RUNG
   RUNG wire#w1
      { S7_Templates := "SrcType := Real"; S7_GenerateENO := "TRUE" } Sub(in1 := "DB26".Dbd8, in2 := "DB26".Dbd12, out => "DB26".Dbd28)
   END_RUNG
   RUNG wire#w1
      { S7_Templates := "SrcType := Real"; S7_GenerateENO := "TRUE" } Sub(in1 := "DB26".Dbd20, in2 := "DB26".Dbd12, out => "DB26".Dbd32)
   END_RUNG
   // the same network as SCL:
   IF "On" THEN
       "DB26".Dbd24 := "DB26".Dbd0 - "DB26".Dbd4;
       "DB26".Dbd28 := "DB26".Dbd8 - "DB26".Dbd12;
       "DB26".Dbd32 := "DB26".Dbd20 - "DB26".Dbd12;
   END_IF;
END_REGION

REGION Network 4: Esegui le operazioni matematiche conclusive
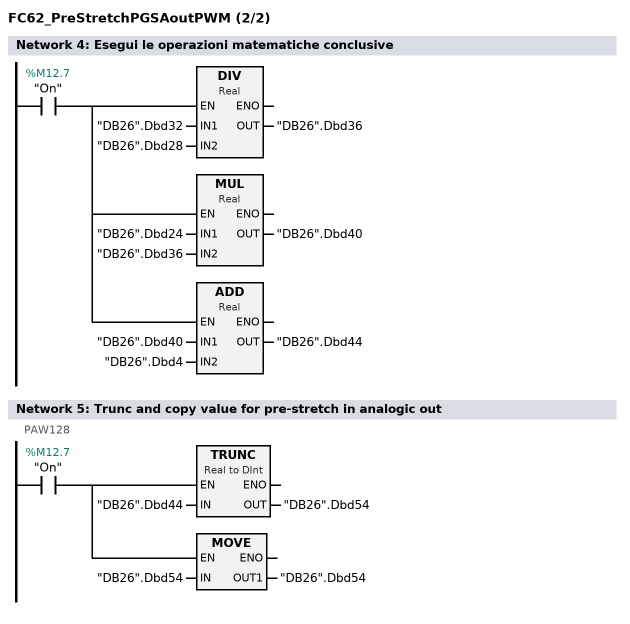
   RUNG wire#powerrail
      Contact( "On" )
      wire#w1
      { S7_Templates := "SrcType := Real"; S7_GenerateENO := "TRUE" } Div(in1 := "DB26".Dbd32, in2 := "DB26".Dbd28, out => "DB26".Dbd36)
   END_RUNG
   RUNG wire#w1
      { S7_Templates := "SrcType := Real"; S7_GenerateENO := "TRUE" } Mul(in1 := "DB26".Dbd24, in2 := "DB26".Dbd36, out => "DB26".Dbd40)
   END_RUNG
   RUNG wire#w1
      { S7_Templates := "SrcType := Real"; S7_GenerateENO := "TRUE" } Add(in1 := "DB26".Dbd40, in2 := "DB26".Dbd4, out => "DB26".Dbd44)
   END_RUNG
   // the same network as SCL:
   IF "On" THEN
       "DB26".Dbd36 := "DB26".Dbd32 / "DB26".Dbd28;
       "DB26".Dbd40 := "DB26".Dbd24 * "DB26".Dbd36;
       "DB26".Dbd44 := "DB26".Dbd40 + "DB26".Dbd4;
   END_IF;
END_REGION

REGION Network 5: Trunc and copy value for pre-stretch in analogic out
   // PAW128
   RUNG wire#powerrail
      Contact( "On" )
      wire#w1
      { S7_Templates := "[SrcType := Real, DestType := DInt]"; S7_GenerateENO := "TRUE" } Trunc(in := "DB26".Dbd44, out => "DB26".Dbd54)
   END_RUNG
   RUNG wire#w1
      { S7_GenerateENO := "TRUE" } Move(in := "DB26".Dbd54, out1 => "DB26".Dbd54)
   END_RUNG
   // the same network as SCL:
   IF "On" THEN
       "DB26".Dbd54 := TRUNC("DB26".Dbd44);
       "DB26".Dbd54 := "DB26".Dbd54;
   END_IF;
END_REGION
END_FUNCTION

FUNCTION "FC63_StretchPGSAoutPWM" : Void   // FC63, LAD
{ S7_Optimized_Access := 'FALSE' }
AUTHOR : PaZan
VERSION : 0.1
// stored: AutoNumber false, IsIECCheckEnabled false, SetENOAutomatically false, UDAEnableTagReadback false
   VAR_TEMP   // added for the SCL form of the ladder/FBD networks
      _w1 : Bool;
   END_VAR
BEGIN

REGION Network 1
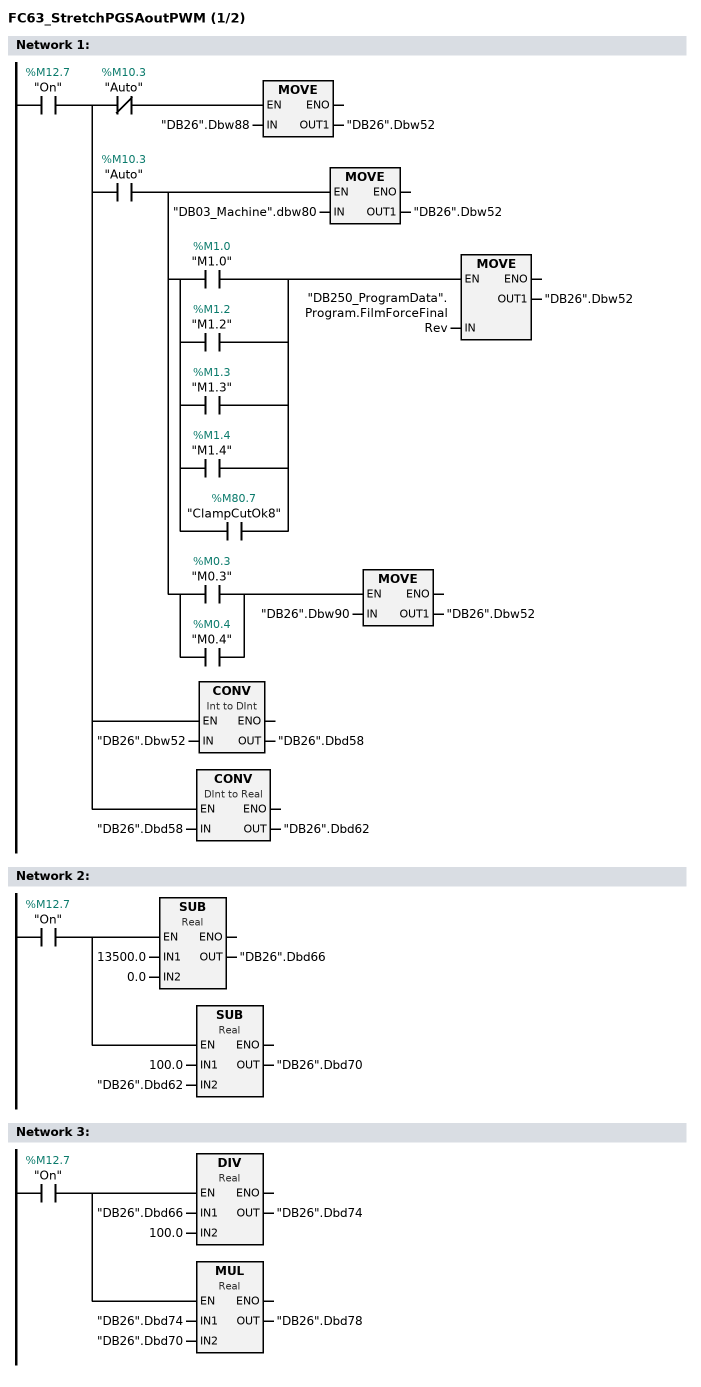
   RUNG wire#powerrail
      Contact( "On" )
      wire#w1
      I_Contact( "Auto" )
      { S7_GenerateENO := "TRUE" } Move(in := "DB26".Dbw88, out1 => "DB26".Dbw52)
   END_RUNG
   RUNG wire#w1
      Contact( "Auto" )
      wire#w2
      { S7_GenerateENO := "TRUE" } Move(in := "DB03_Machine".dbw80, out1 => "DB26".Dbw52)
   END_RUNG
   RUNG wire#w2
      Contact( "M1.0" )
      wire#w3
      { S7_GenerateENO := "TRUE" } Move(in := "DB250_ProgramData".Program.FilmForceFinalRev, out1 => "DB26".Dbw52)
   END_RUNG
   RUNG wire#w2
      Contact( "M1.2" )
   END_RUNG wire#w3
   RUNG wire#w2
      Contact( "M1.3" )
   END_RUNG wire#w3
   RUNG wire#w2
      Contact( "M1.4" )
   END_RUNG wire#w3
   RUNG wire#w2
      Contact( "ClampCutOk8" )
   END_RUNG wire#w3
   RUNG wire#w2
      Contact( "M0.3" )
      wire#w4
      { S7_GenerateENO := "TRUE" } Move(in := "DB26".Dbw90, out1 => "DB26".Dbw52)
   END_RUNG
   RUNG wire#w2
      Contact( "M0.4" )
   END_RUNG wire#w4
   RUNG wire#w1
      { S7_Templates := "[SrcType := Int, DestType := DInt]"; S7_GenerateENO := "TRUE" } Convert(in := "DB26".Dbw52, out => "DB26".Dbd58)
   END_RUNG
   RUNG wire#w1
      { S7_Templates := "[SrcType := DInt, DestType := Real]"; S7_GenerateENO := "TRUE" } Convert(in := "DB26".Dbd58, out => "DB26".Dbd62)
   END_RUNG
   // the same network as SCL:
   IF "On" AND NOT "Auto" THEN "DB26".Dbw52 := "DB26".Dbw88; END_IF;
   #_w1 := "On" AND "Auto";
   IF #_w1 THEN "DB26".Dbw52 := "DB03_Machine".dbw80; END_IF;
   IF #_w1 AND ("M1.0" OR "M1.2" OR "M1.3" OR "M1.4" OR "ClampCutOk8") THEN
       "DB26".Dbw52 := "DB250_ProgramData".Program.FilmForceFinalRev;
   END_IF;
   IF #_w1 AND ("M0.3" OR "M0.4") THEN "DB26".Dbw52 := "DB26".Dbw90; END_IF;
   IF "On" THEN
       "DB26".Dbd58 := INT_TO_DINT("DB26".Dbw52);
       "DB26".Dbd62 := DINT_TO_REAL("DB26".Dbd58);
   END_IF;
END_REGION

REGION Network 2
   RUNG wire#powerrail
      Contact( "On" )
      wire#w1
      { S7_Templates := "SrcType := Real"; S7_GenerateENO := "TRUE" } Sub(in1 := 13500.0, in2 := 0.0, out => "DB26".Dbd66)
   END_RUNG
   RUNG wire#w1
      { S7_Templates := "SrcType := Real"; S7_GenerateENO := "TRUE" } Sub(in1 := 100.0, in2 := "DB26".Dbd62, out => "DB26".Dbd70)
   END_RUNG
   // the same network as SCL:
   IF "On" THEN
       "DB26".Dbd66 := 13500.0 - 0.0;
       "DB26".Dbd70 := 100.0 - "DB26".Dbd62;
   END_IF;
END_REGION

REGION Network 3
   RUNG wire#powerrail
      Contact( "On" )
      wire#w1
      { S7_Templates := "SrcType := Real"; S7_GenerateENO := "TRUE" } Div(in1 := "DB26".Dbd66, in2 := 100.0, out => "DB26".Dbd74)
   END_RUNG
   RUNG wire#w1
      { S7_Templates := "SrcType := Real"; S7_GenerateENO := "TRUE" } Mul(in1 := "DB26".Dbd74, in2 := "DB26".Dbd70, out => "DB26".Dbd78)
   END_RUNG
   // the same network as SCL:
   IF "On" THEN
       "DB26".Dbd74 := "DB26".Dbd66 / 100.0;
       "DB26".Dbd78 := "DB26".Dbd74 * "DB26".Dbd70;
   END_IF;
END_REGION

REGION Network 4: Trunc and copy value for stretch torque in analogic out
   // PAW130
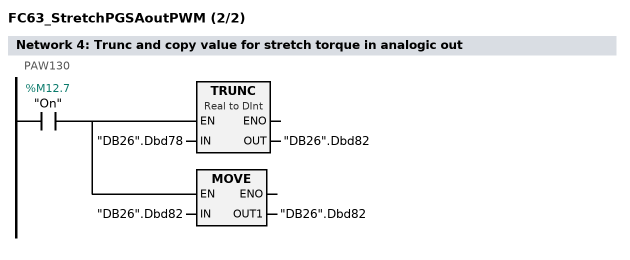
   RUNG wire#powerrail
      Contact( "On" )
      wire#w1
      { S7_Templates := "[SrcType := Real, DestType := DInt]"; S7_GenerateENO := "TRUE" } Trunc(in := "DB26".Dbd78, out => "DB26".Dbd82)
   END_RUNG
   RUNG wire#w1
      { S7_GenerateENO := "TRUE" } Move(in := "DB26".Dbd82, out1 => "DB26".Dbd82)
   END_RUNG
   // the same network as SCL:
   IF "On" THEN
       "DB26".Dbd82 := TRUNC("DB26".Dbd78);
       "DB26".Dbd82 := "DB26".Dbd82;
   END_IF;
END_REGION
END_FUNCTION

FUNCTION_BLOCK "SINA_SPEED_Motor_Centrador"
TITLE = 'Speed Control with SINAMICS and S7'
{ S7_Optimized_Access := 'TRUE' }
AUTHOR : DRVDPS7
FAMILY : DRIVES
NAME : SINA_SPD
VERSION : 5.1
//Copyright (C) Siemens AG 2012. All Rights Reserved. Confidential
//-------------------------------------------------------------------------------------- 
//SINA_SPEED: Drehzahlregelung mit dem Antriebsbaustein SINAMICS S120/G120 <-> S7-1200
//------------------------------------------------------------------------------------- Ersteller: Siemens AG Erlangen A&D MC PM   Datum:  07.07.10        Vers.:2.1
//Änderung:  J.B. Typical Team                       07.12.12              2.2
//    Umsetzung in SCL / TIA 
//Änderung:  J.B. Typical Team                       29.04.13              2.3
//    1. "Q" an den AusgÃ¤nge entfernen
//    2. Neuer Ausgang PwrInhibit
//Änderung:  J.B. Typical Team                       28.06.13              2.4
//    Ã„nderung HW-Zugriff Ã¼ber LOG2MOD
//     
//Änderung:  J.B. Typical Team                       18.07.13              2.5
//    Ã„nderung HW-Zugriff Ã¼ber zwei HW-EingÃ¤nge
//
//Änderung:  J.B. Typical Team                       17.07.14              3.0
//    Optimmierung
//
//Änderung:  J.B. Typical Team                       30.07.14              4.0
//    Festlegung auf einheitlicher neuer Version 4.0
//
//Änderung:  P.Z. Typical Team                       03.12.15              4.1
//    Schnittstelle an Programmierleitfadeb TIA-Potal angepasst
//    zusÃ¤tzlicher Eingang "ConfigAxis" fÃ¼r STW-Bits
//
//Änderung:  G.F. Typical Team                       01.03.16              4.2
//    Sollwert auf INT - Grenzen begrenzt
//Änderung:  F.G. Typical Team                       13.09.16              4.3
//    Ausgabewerte am Ausgang "Status" angepasst 
//
//Änderung:  G.F. Typical Team                       11.01.17              5.0
//    - Festlegung auf einheitlicher neuer Version 5.0 
//
//Änderung:  G.F. Typical Team                       03.05.18              5.1
//    - Alle Bits des Eingang ConfigAxis auf STW1 aufgelegt 
//
//Bibliothek V7
//Funktion: Drehzahlregelung mit dem Antriebsbaustein SINAMICS S120/G120 <-> S7-1200
//********************************************************************************************************************************************************
//************************************************************************FB283***************************************************************************
//********************************************************************************************************************************************************
   VAR_INPUT 
      EnableAxis : Bool := 0;   // 0-->1; 1 = Enable the drive (OFF2 / OFF 3 are 1 in default status) (OFF1 = 0-->1)
      AckError : Bool := 0;   // 1 = Acknowledge drive error
      SpeedSp : Real := 0.0;   // Speed standardises with the standardisation factor
      RefSpeed : Real := 0.0;   // Standardisation factor of speed
      ConfigAxis : Word := 16#003F;   // binary programmed input to control all functions in the telegram without its own function block input
      HWIDSTW : HW_IO := 0;   // Hardware Identifer set point slot
      HWIDZSW : HW_IO := 0;   // Hardware Identifer actual value slot
   END_VAR

   VAR_OUTPUT 
      AxisEnabled : Bool := 0;   // 1 = Drive is enabled
      Lockout : Bool := 0;   // 1 = Drive lockout active
      ActVelocity : Real := 0.0;   // Actual in [U/min]
      Error : Bool := 0;   // 1 = Error  (FB and Infeed)
      Status : Word := 0;   // Status output (7002 = FB in operation; 8xxx = error description  - read the manual)
      DiagId : Word := 16#0000;   // Error codes of the cyclic system funtion blocks DPWR / DPRD_DAT
   END_VAR

   VAR 
      sxSendBuf : Struct   // Send buffer
         STW1 : Word := WORD#16#0000;   // STW1sxSTW1     : STRUCT            Bit08       : BOOL:=False;              // ST-Wort-1 Bit 08 --> Reserve            Bit09       : BOOL:=False;              // ST-Wort-1 Bit 09 --> Reserve            Bit10       : BOOL:=True;               // ST-Wort-1 Bit 10 --> FÃ¼hrung durch PLC            Dir         : BOOL:=False;              // ST-Wort-1 Bit 11 --> Direction            Bit12       : BOOL:=False;              // ST-Wort-1 Bit 12 --> Haltebremse unbedingt Ã¶ffnen            Bit13       : BOOL:=False;              // ST-Wort-1 Bit 13 --> Motorpotenziometer Sollwert hÃ¶her            Bit14       : BOOL:=False;              // ST-Wort-1 Bit 14 --> Motorpotenziometer Sollwert tiefer            Bit15       : BOOL:=False;              // ST-Wort-1 Bit 15 --> Reserviert            Off1        : BOOL:=False;              // ST-Wort-1 Bit 00 --> OFF1/ON (flanks acceptance)            Off2        : BOOL:=True;               // ST-Wort-1 Bit 01 --> OFF2/ON (enable possible)            Off3        : BOOL:=True;               // ST-Wort-1 Bit 02 --> OFF3/ON (enable possible)            InvEn       : BOOL:=True;               // ST-Wort-1 Bit 03 --> Enable controller            RampEn      : BOOL:=True;               // ST-Wort-1 Bit 04 --> Ramp enable            RampOn      : BOOL:=True;               // ST-Wort-1 Bit 05 --> Ramp On            SpEn        : BOOL:=True;               // ST-Wort-1 Bit 06 --> Speed set point enable            AckFlt      : BOOL:=False;              // ST-Wort-1 Bit 07 --> Acknowledge fault         END_STRUCT;
         Velocity : Word := WORD#16#0000;   // Setpoint of velocity
      END_STRUCT;
      sxRecvBuf : Struct   // Receive buffer
         ZSW1 : Word := WORD#16#0000;   // ZSW1sxZSW1     : STRUCT            SpDev       : BOOL:=False;              // ZSW-Wort-1 = Schleppfehler im Toleranzbereich            Pcd         : BOOL:=False;              // ZSW-Wort-1 = PZD-FÃ¼hrung erreicht            Comp        : BOOL:=False;              // ZSW-Wort-1 = Zielposition erreicht            CurLim      : BOOL:=False;              // ZSW-Wort-1 = Referenzpunkt gesetzt            Brake       : BOOL:=False;              // ZSW-Wort-1 = Haltebremse Ã¶ffnen            Motover     : BOOL:=False;              // ZSW-Wort-1 = keine Warnung Ãœbertemperatur Motor            Dir         : BOOL:=False;              // ZSW-Wort-1 = Direction            Invover     : BOOL:=False;              // ZSW-Wort-1 = keine Warnung thermische Ãœberlast Leistungsteil            Rts         : BOOL:=False;              // ZSW-Wort-1 = Ready to power up / to start            Rdy         : BOOL:=False;              // ZSW-Wort-1 = Ready to operate            IOp         : BOOL:=False;              // ZSW-Wort-1 = In operation (operation enabled)            Fault       : BOOL:=False;              // ZSW-Wort-1 = Fault present            NoOff2      : BOOL:=False;              // ZSW-Wort-1 = OFF2 inactive            NoOff3      : BOOL:=False;              // ZSW-Wort-1 = OFF3 inactive            Inhibit     : BOOL:=False;              // ZSW-Wort-1 = Power ON inhibit active             Alarm       : BOOL:=False;              // ZSW-Wort-1 = Alarm / Warning present                     END_STRUCT;
         Velocity : Word := WORD#16#0000;   // Feedback of velocity
      END_STRUCT;
   END_VAR

   VAR_TEMP 
      piRetSFC : Int;   // Status for fault analysis
      piCount : Int;   // Freely available counter variable 3
      prVelocity : Real;   // velocity
      pdRecvBuf : DWord;   // Buffer of Recv-Value
      pdSendBuf : DWord;   // Buffer of Send-Value
      phLAddr : HW_IO;   // Start addr from the I/O process image area of mod (DEC) for DPWR_DAT/DPRD_DAT
      swSendBuf : Array[0..1] of Word;   // Sendepuffer
      swRecvBuf : Array[0..1] of Word;   // Empfangspuffer         Static variables
   END_VAR


BEGIN
	
	//=============================================================================
	//SIEMENS AG
	//(c)Copyright 2017 All Rights Reserved
	//-----------------------------------------------------------------------------
	// Library: DriveLib
	// Tested with: S7-1516-3 PN/DP V1.8
	// Engineering: TIA Portal V14
	// Restrictions: -
	// Requirements: S7-1200 / S7-1500
	// Functionality: cyclic communication between a SINAMICS a PLC.
	//                If in HWConfig Std.TLG 1 is projected 2 PZD-words are exchanged
	//                in every bus cycle.
	//                The parametrisation of these words is described in the manual of the
	//                SINAMICS
	//=============================================================================
	
	// Schreibdaten zusammenstellen
	// Steuerword aufbereiten
	
	#sxSendBuf.STW1.%X0 := #EnableAxis;
	#sxSendBuf.STW1.%X1 := #ConfigAxis.%X0;
	#sxSendBuf.STW1.%X2 := #ConfigAxis.%X1;
	#sxSendBuf.STW1.%X3 := #ConfigAxis.%X2;
	#sxSendBuf.STW1.%X4 := #ConfigAxis.%X3;
	#sxSendBuf.STW1.%X5 := #ConfigAxis.%X4;
	#sxSendBuf.STW1.%X6 := #ConfigAxis.%X5;
	#sxSendBuf.STW1.%X7 := #AckError;
	#sxSendBuf.STW1.%X8 := #ConfigAxis.%X10;
	#sxSendBuf.STW1.%X9 := #ConfigAxis.%X11;
	#sxSendBuf.STW1.%X10 := TRUE;
	#sxSendBuf.STW1.%X11 := #ConfigAxis.%X6;
	#sxSendBuf.STW1.%X12 := #ConfigAxis.%X7;
	#sxSendBuf.STW1.%X13 := #ConfigAxis.%X8;
	#sxSendBuf.STW1.%X14 := #ConfigAxis.%X9;
	#sxSendBuf.STW1.%X15 := #ConfigAxis.%X12;
	
	// Geschwindigkeit
	IF #RefSpeed <> 0 THEN
	  #prVelocity := #SpeedSp * (16384.0 / #RefSpeed);
	  // Limit REAL - Variable to INT - Limits
	  IF #prVelocity > 32767 THEN
	    #prVelocity := 32767;
	  ELSIF #prVelocity < -32768 THEN
	    #prVelocity := -32768;
	  ELSE
	    ; // not needed
	  END_IF;
	  #sxSendBuf.Velocity := INT_TO_WORD(REAL_TO_INT(#prVelocity));
	  
	ELSE
	  #sxSendBuf.Velocity := W#16#0;
	END_IF;
	#swSendBuf[0] := #sxSendBuf.STW1;
	#swSendBuf[1] := #sxSendBuf.Velocity;
	
	//Prozessdaten zur Signalbaugruppe schreiben
	#piRetSFC := DPWR_DAT(LADDR := #HWIDSTW,
	                      RECORD := #swSendBuf);
	
	// Fehler der RÃ¼ckmeldung ausgeben
	#DiagId := INT_TO_WORD(#piRetSFC);
	
	//kein Fehler beim Schreiben
	IF #piRetSFC = 0 THEN
	  
	  //kein Fehler beim Schreiben
	  IF #piRetSFC = 0 THEN
	    
	    //Prozessdaten von der Signalbaugruppe lesen
	    #piRetSFC := DPRD_DAT(LADDR := #HWIDZSW,
	                          RECORD => #swRecvBuf);
	    
	    // Fehler der RÃ¼ckmeldung ausgeben
	    #DiagId := INT_TO_WORD(#piRetSFC);
	  END_IF;
	  
	  //Fehler beim Lesen (Profibus-Kommunikation unterbrochen)
	  IF #piRetSFC <> 0 THEN
	    
	    // Fehler
	    #Error := TRUE;
	    #Status := 16#8600;
	    
	    // Zustandsworte lÃ¶schen
	    #sxRecvBuf.ZSW1.%X8 := 0;
	    #sxRecvBuf.ZSW1.%X9 := 0;
	    #sxRecvBuf.ZSW1.%X10 := 0;
	    #sxRecvBuf.ZSW1.%X11 := 0;
	    #sxRecvBuf.ZSW1.%X12 := 0;
	    #sxRecvBuf.ZSW1.%X13 := 0;
	    #sxRecvBuf.ZSW1.%X14 := 0;
	    #sxRecvBuf.ZSW1.%X15 := 0;
	    #sxRecvBuf.ZSW1.%X0 := 0;
	    #sxRecvBuf.ZSW1.%X1 := 0;
	    #sxRecvBuf.ZSW1.%X2 := 0;
	    #sxRecvBuf.ZSW1.%X3 := 0;
	    #sxRecvBuf.ZSW1.%X4 := 0;
	    #sxRecvBuf.ZSW1.%X5 := 0;
	    #sxRecvBuf.ZSW1.%X6 := 0;
	    #sxRecvBuf.ZSW1.%X7 := 0;
	    
	    
	    (*#sxRecvBuf.sxZSW1.SpDev   := 0;
	    #sxRecvBuf.sxZSW1.Pcd     := 0;
	    #sxRecvBuf.sxZSW1.Comp    := 0;
	    #sxRecvBuf.sxZSW1.CurLim  := 0;
	    #sxRecvBuf.sxZSW1.Brake   := 0;
	    #sxRecvBuf.sxZSW1.Motover := 0;
	    #sxRecvBuf.sxZSW1.Dir     := 0;
	    #sxRecvBuf.sxZSW1.Invover := 0;
	    #sxRecvBuf.sxZSW1.Rts     := 0;
	    #sxRecvBuf.sxZSW1.Rdy     := 0;
	    #sxRecvBuf.sxZSW1.IOp     := 0;
	    #sxRecvBuf.sxZSW1.Fault   := 0;
	    #sxRecvBuf.sxZSW1.NoOff2  := 0;
	    #sxRecvBuf.sxZSW1.NoOff3  := 0;
	    #sxRecvBuf.sxZSW1.Inhibit := 0;
	    #sxRecvBuf.sxZSW1.Alarm   := 0;*)
	    
	    #sxRecvBuf.Velocity := W#16#00;
	    
	    // Werte auslesen
	  ELSE
	    #sxRecvBuf.ZSW1 := #swRecvBuf[0];
	    #sxRecvBuf.Velocity := #swRecvBuf[1];
	    
	    // ZSW1 aufbereiten                       
	    #AxisEnabled := #sxRecvBuf.ZSW1.%X2;
	    #Error := #sxRecvBuf.ZSW1.%X3 OR #sxRecvBuf.ZSW1.%X6;
	    #Lockout := #sxRecvBuf.ZSW1.%X6;
	    
	    // Fehler auswerten
	    IF #sxRecvBuf.ZSW1.%X3 THEN
	      #Status := 16#8401;
	    ELSIF #sxRecvBuf.ZSW1.%X6 THEN
	      #Status := 16#8402;
	    ELSE
	      #Status := 16#7002;
	    END_IF;
	    
	    (*#Busy       := #sxRecvBuf.sxZSW1.IOp;
	    #Error      := #sxRecvBuf.sxZSW1.Fault OR #sxRecvBuf.sxZSW1.Inhibit;
	    #PwrInhibit := #sxRecvBuf.sxZSW1.Inhibit;            
	
	    // Fehler auswerten
	    IF #sxRecvBuf.sxZSW1.Fault THEN
	        #ErrorId := 1;
	    ELSIF #sxRecvBuf.sxZSW1.Inhibit THEN 
	        #ErrorId := 2;
	    ELSE
	        #ErrorId := 0;    
	    END_IF;*)
	    
	    // Geschwindigkeit
	    IF #RefSpeed <> 0 THEN
	      #ActVelocity := INT_TO_REAL(WORD_TO_INT(#sxRecvBuf.Velocity)) / (16384.0 / #RefSpeed);
	    ELSE
	      #ActVelocity := 0.0;
	    END_IF;
	  END_IF;
	ELSE
	  
	  // Fehler
	  #Error := TRUE;
	  #Status := 16#8601;
	  
	END_IF;
	
	
	
END_FUNCTION_BLOCK

DATA_BLOCK "Centrador_Paletes_DB"   // DB11
VERSION : 0.1
// stored: AutoNumber true, InstanceOfName Centrador_Paletes, InstanceOfType FB
"Centrador_Paletes"
BEGIN
END_DATA_BLOCK

DATA_BLOCK "Modbus_DB"   // DB28
VERSION : 0.1
// stored: AutoNumber false, InstanceOfName Modbus, InstanceOfType FB
"Modbus"
BEGIN
END_DATA_BLOCK

DATA_BLOCK "SINA_SPEED_Motor_Centrador_DB"   // DB11
AUTHOR : DRVDPS7
FAMILY : DRIVES
NAME : SINA_SPD
VERSION : 5.1
// stored: AutoNumber true, InstanceOfName SINA_SPEED_Motor_Centrador, InstanceOfType FB
"SINA_SPEED_Motor_Centrador"
BEGIN
END_DATA_BLOCK

DATA_BLOCK "U201_Process_Data"   // DB211
VERSION : 0.1
// stored: AutoNumber false, InstanceOfName Inverter_Process_Data, InstanceOfType FB
"Inverter_Process_Data"
BEGIN
END_DATA_BLOCK

DATA_BLOCK "U221_Process_Data"   // DB212
VERSION : 0.1
// stored: AutoNumber false, InstanceOfName Inverter_Process_Data, InstanceOfType FB
"Inverter_Process_Data"
BEGIN
END_DATA_BLOCK

DATA_BLOCK "U241_Process_Data"   // DB213
VERSION : 0.1
// stored: AutoNumber false, InstanceOfName Inverter_Process_Data, InstanceOfType FB
"Inverter_Process_Data"
BEGIN
END_DATA_BLOCK

DATA_BLOCK "EncoderCh0-CarriageA"   // DB102
// stored: AutoNumber false, InstanceOfName CTRL_HSC, OfSystemLibElement CTRL_HSC, OfSystemLibVersion 1.0
"CTRL_HSC"
   // VAR_INPUT
   //    HSC : HW_HSC;
   //    DIR : Bool;
   //    CV : Bool;
   //    RV : Bool;
   //    PERIOD : Bool;
   //    NEW_DIR : Int;
   //    NEW_CV : DInt;
   //    NEW_RV : DInt;
   //    NEW_PERIOD : Int;
   // END_VAR
   // VAR_OUTPUT
   //    BUSY : Bool;
   //    STATUS : Word;
   // END_VAR
BEGIN
END_DATA_BLOCK

DATA_BLOCK "EncoderCh1-CarriageB"   // DB103
// stored: AutoNumber false, InstanceOfName CTRL_HSC, OfSystemLibElement CTRL_HSC, OfSystemLibVersion 1.0
"CTRL_HSC"
   // VAR_INPUT
   //    HSC : HW_HSC;
   //    DIR : Bool;
   //    CV : Bool;
   //    RV : Bool;
   //    PERIOD : Bool;
   //    NEW_DIR : Int;
   //    NEW_CV : DInt;
   //    NEW_RV : DInt;
   //    NEW_PERIOD : Int;
   // END_VAR
   // VAR_OUTPUT
   //    BUSY : Bool;
   //    STATUS : Word;
   // END_VAR
BEGIN
END_DATA_BLOCK

DATA_BLOCK "IEC_Timer_0_DB"   // DB15
{ S7_Optimized_Access := 'TRUE' }
// stored: AutoNumber true, InstanceOfName IEC_TIMER, OfSystemLibElement IEC_TIMER, OfSystemLibVersion 1.0
"IEC_TIMER"
   // VAR
   //    PT : Time;
   //    ET { ExternalWritable := 'False'} : Time;
   //    IN : Bool;
   //    Q { ExternalWritable := 'False'} : Bool;
   // END_VAR
BEGIN
END_DATA_BLOCK
